(* PLC project Rasi_feeds_batching.project, Automation Builder 2.7 - Basic Automation Builder 2.7 *)
(* stored: creationDateTime 2026-08-27T18:20:00 *)

PROGRAM test_fbd_boxes
  VAR
    Auto_Ctrl : Auto_Batching_V14;
    Semi_Auto_Ctrl : Semi_Auto_Batching_V14;
  END_VAR

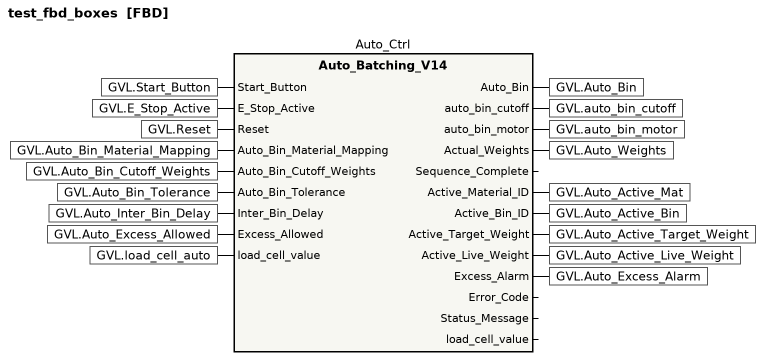
(* FBD diagram, written out as Structured Text *)
Auto_Ctrl(Start_Button := GVL.Start_Button, E_Stop_Active := GVL.E_Stop_Active, Reset := GVL.Reset, Auto_Bin_Material_Mapping := GVL.Auto_Bin_Material_Mapping, Auto_Bin_Cutoff_Weights := GVL.Auto_Bin_Cutoff_Weights, Auto_Bin_Tolerance := GVL.Auto_Bin_Tolerance, Inter_Bin_Delay := GVL.Auto_Inter_Bin_Delay, Excess_Allowed := GVL.Auto_Excess_Allowed, load_cell_value := GVL.load_cell_auto);
GVL.Auto_Bin := Auto_Ctrl.Auto_Bin;
GVL.auto_bin_cutoff := Auto_Ctrl.auto_bin_cutoff;
GVL.auto_bin_motor := Auto_Ctrl.auto_bin_motor;
GVL.Auto_Weights := Auto_Ctrl.Actual_Weights;
GVL.Auto_Active_Mat := Auto_Ctrl.Active_Material_ID;
GVL.Auto_Active_Bin := Auto_Ctrl.Active_Bin_ID;
GVL.Auto_Active_Target_Weight := Auto_Ctrl.Active_Target_Weight;
GVL.Auto_Active_Live_Weight := Auto_Ctrl.Active_Live_Weight;
GVL.Auto_Excess_Alarm := Auto_Ctrl.Excess_Alarm;
END_PROGRAM
